FUNCTION_BLOCK FB_StationStats
VAR_INPUT
	iLoading:BOOL;
	iUnloading:BOOL;
	iBlocked:BOOL;
	iStarved:BOOL;
	iWaitAux:BOOL;
	
END_VAR
VAR_OUTPUT
	qStationState:enumStationState;
END_VAR
VAR
	tLoadingTime:UINT;
	tCyclingTime:UINT;
	tUnloadingTime:UINT;
	tBlockedTime:UINT;
	tStarvedTime:UINT;
	tWaitAuxTime:UINT;
	tFaultTime:UINT;
	tRepairTime:UINT;
	
	tTotalCycleTime:UINT;
	
	tNotCycle: BOOL;
	tAnyButtonPressed: BOOL;
	
	osrResetTime:F_TRIG;
	tFaultLockout: BOOL;
	
	osrClearRepair:R_TRIG;
	timedelayCycleCheck:TOF;
END_VAR
VAR_IN_OUT
		stndata:typeStation;
END_VAR

//timer block for recording machine states

IF gHMIButtons.gAnyButtonPressed AND stndata.Data.Fault THEN
	tAnyButtonPressed := TRUE;
END_IF

//work out if is cycle time
IF iLoading OR iUnloading OR iBlocked OR iStarved OR iWaitAux  THEN
	tNotCycle := TRUE;
	ELSE
	tNotCycle := FALSE;
END_IF

//auto cycle timer
IF stndata.Data.AutoCycling AND NOT tNotCycle AND NOT tFaultLockout  THEN
	IF System.PulseHundredMilliSecond THEN
		tCyclingTime := tCyclingTime + 1;
	END_IF
	qStationState := enumStationState.Cycling;
END_IF

//Loading cycle timer
IF iLoading AND NOT tFaultLockout THEN
	IF System.PulseHundredMilliSecond THEN
		tLoadingTime := tLoadingTime + 1;
	END_IF
	qStationState := enumStationState.Loading;
END_IF

//Unloading cycle timer
IF iUnloading AND NOT tFaultLockout THEN
	IF System.PulseHundredMilliSecond THEN
		tUnloadingTime := tUnloadingTime + 1;
	END_IF
	qStationState := enumStationState.Unloading;
END_IF

//blocked cycle timer
IF iBlocked AND NOT tFaultLockout  THEN
	IF System.PulseHundredMilliSecond THEN
		tBlockedTime := tBlockedTime + 1;
	END_IF
	qStationState := enumStationState.Blocked;
END_IF

//starved cycle timer
IF iStarved AND NOT tFaultLockout THEN
	IF System.PulseHundredMilliSecond THEN
		tStarvedTime := tStarvedTime + 1;
	END_IF
	qStationState := enumStationState.Starved;
END_IF

//debounce by a time to capture state change
timedelayCycleCheck(IN:=stndata.Data.AutoCycling,PT:=T#100MS);

//fault cycle timer
//capture time when autocycle ceases and stop counting when a button is pressed, indicating someone is aware of it
IF stndata.Data.Fault AND (timedelayCycleCheck.Q OR tFaultLockout) AND NOT tAnyButtonPressed THEN
	IF System.PulseHundredMilliSecond THEN
		tFaultTime := tFaultTime + 1;
	END_IF
	tFaultLockout := TRUE;
	qStationState := enumStationState.Faulted;
END_IF

//repair time cycle timer
//if anyone has pressed any button during the fault state, then someone is aware it need to be repaired
IF tFaultLockout AND tAnyButtonPressed THEN
	IF System.PulseHundredMilliSecond THEN
		tRepairTime := tRepairTime + 1;
	END_IF
	qStationState := enumStationState.Repair;
END_IF

osrClearRepair(CLK:=stndata.Data.AutoCycling);
IF osrClearRepair.Q THEN
	tFaultLockout := FALSE;
	tAnyButtonPressed := FALSE;
END_IF

//add up to get cycle time
tTotalCycleTime := 		tLoadingTime +	
						tCyclingTime + 
						tUnloadingTime +
						tBlockedTime +
						tStarvedTime + 
						tWaitAuxTime +
						tFaultTime
						;

//reset timer on edge of unloading
osrResetTime(CLK := iUnloading);

IF osrResetTime.Q THEN
	actClearCounters();
END_IF

ACTION actClearCounters:
tLoadingTime		:= 0;
tCyclingTime		:= 0;
tUnloadingTime		:= 0;
tBlockedTime		:= 0;
tStarvedTime		:= 0;
tWaitAuxTime		:= 0;
tFaultTime			:= 0;
END_ACTION

END_FUNCTION_BLOCK

(* stored: Version 1.1.0.1, ProductVersion 3.1.4024.11
   POU FB_StationStats: Id {a386013d-f36c-0689-0762-bfe760851d2d}, SpecialFunc None
   Action actClearCounters: Id {15a985f2-2111-0b31-39fc-1dfb144a9c12} *)
